{attribute 'GeneratedUsingTerminal: EL2262-0000-0004'}
{attribute addProperty BoxType "EL2262-0000-0004"}
{attribute addProperty Id "EtcSlaveTerminalBaseStartTimeNextOutputAT %I*StartTimeNextOutput_228767F44CycCount0AT %Q*CycCount0_AF431CE02Sample0_0AT %Q*Sample_0023574C1Sample0_1AT %Q*Sample_0023574C1Sample0_2AT %Q*Sample_0023574C1Sample0_3AT %Q*Sample_0023574C1Sample0_4AT %Q*Sample_0023574C1Sample0_5AT %Q*Sample_0023574C1Sample0_6AT %Q*Sample_0023574C1Sample0_7AT %Q*Sample_0023574C1Sample0_8AT %Q*Sample_0023574C1Sample0_9AT %Q*Sample_0023574C1GapAT %I*EMPTY_STRUCTURE0CycCount1AT %Q*CycCount1_A8B5FFE62Sample1_0AT %Q*Sample_07D5B44A1Sample1_1AT %Q*Sample_07D5B44A1Sample1_2AT %Q*Sample_07D5B44A1Sample1_3AT %Q*Sample_07D5B44A1Sample1_4AT %Q*Sample_07D5B44A1Sample1_5AT %Q*Sample_07D5B44A1Sample1_6AT %Q*Sample_07D5B44A1Sample1_7AT %Q*Sample_07D5B44A1Sample1_8AT %Q*Sample_07D5B44A1Sample1_9AT %Q*Sample_07D5B44A1Gap_1AT %I*EMPTY_STRUCTURE0WcStateAT %I*WcState_9091E0EB2InfoDataAT %I*InfoData_A7436BC610"}
{attribute addProperty CRC "1537807177"}
{attribute addProperty Size "40"}
TYPE EL2262_5BA91349 EXTENDS EtcSlaveTerminalBase :
STRUCT
	{attribute addProperty Name "StartTimeNextOutput"}
	StartTimeNextOutput : StartTimeNextOutput_228767F4;
	{attribute addProperty Name "CycCount0"}
	CycCount0 : CycCount0_AF431CE0;
	{attribute addProperty Name "Sample0_0"}
	Sample0_0 : Sample_0023574C;
	{attribute addProperty Name "Sample0_1"}
	Sample0_1 : Sample_0023574C;
	{attribute addProperty Name "Sample0_2"}
	Sample0_2 : Sample_0023574C;
	{attribute addProperty Name "Sample0_3"}
	Sample0_3 : Sample_0023574C;
	{attribute addProperty Name "Sample0_4"}
	Sample0_4 : Sample_0023574C;
	{attribute addProperty Name "Sample0_5"}
	Sample0_5 : Sample_0023574C;
	{attribute addProperty Name "Sample0_6"}
	Sample0_6 : Sample_0023574C;
	{attribute addProperty Name "Sample0_7"}
	Sample0_7 : Sample_0023574C;
	{attribute addProperty Name "Sample0_8"}
	Sample0_8 : Sample_0023574C;
	{attribute addProperty Name "Sample0_9"}
	Sample0_9 : Sample_0023574C;
	{attribute addProperty Name "Gap"}
	Gap : EMPTY_STRUCTURE;
	{attribute addProperty Name "CycCount1"}
	CycCount1 : CycCount1_A8B5FFE6;
	{attribute addProperty Name "Sample1_0"}
	Sample1_0 : Sample_07D5B44A;
	{attribute addProperty Name "Sample1_1"}
	Sample1_1 : Sample_07D5B44A;
	{attribute addProperty Name "Sample1_2"}
	Sample1_2 : Sample_07D5B44A;
	{attribute addProperty Name "Sample1_3"}
	Sample1_3 : Sample_07D5B44A;
	{attribute addProperty Name "Sample1_4"}
	Sample1_4 : Sample_07D5B44A;
	{attribute addProperty Name "Sample1_5"}
	Sample1_5 : Sample_07D5B44A;
	{attribute addProperty Name "Sample1_6"}
	Sample1_6 : Sample_07D5B44A;
	{attribute addProperty Name "Sample1_7"}
	Sample1_7 : Sample_07D5B44A;
	{attribute addProperty Name "Sample1_8"}
	Sample1_8 : Sample_07D5B44A;
	{attribute addProperty Name "Sample1_9"}
	Sample1_9 : Sample_07D5B44A;
	{attribute addProperty Name "Gap_1"}
	Gap_1 : EMPTY_STRUCTURE;
	{attribute addProperty Name "WcState"}
	WcState : WcState_9091E0EB;
	{attribute addProperty Name "InfoData"}
	InfoData : InfoData_A7436BC6;
END_STRUCT
END_TYPE

(* stored: Version 1.2.0.0, ProductVersion 3.1.4024.9
   DUT EL2262_5BA91349: Id {5e480338-dd5a-4df6-83e6-039c365eec76} *)
